(*			
	RAFALOS
	Rafał Osajda		19.09.2025		TC 4024.66
	Komponent bazowy dla elementów prostych
*)
FUNCTION_BLOCK FB_BaseComponent EXTENDS FB_BaseLoggerElement IMPLEMENTS ITF_BaseComponent, ITF_BaseComponent_HMI_Connector
VAR
	cmdReset						: FB_BaseCommand;
	cmdParametersCreate				: FB_BaseCommand;
	cmdParametersRestoreToDefault	: FB_BaseCommand;
	
	
END_VAR
VAR PERSISTENT
	stParameters					: ST_Parameters;
END_VAR

(*			
	RafalOS
	Rafał Osajda		27.03.2025		TC 4024.66
	Obsluga bledow sprawdzanie czy jakis blad sie nei pojawil i ustawienie stanu lub wylaczenie
*)
METHOD PUBLIC ExecuteEveryCycle_Error
VAR_INPUT
END_VAR
END_METHOD

(*			
	RafalOS
	Rafał Osajda		27.03.2025		TC 4024.66
	Wywolanie co cykl operacji 
*)
METHOD PUBLIC ExecuteEveryCycle_Operation
VAR_INPUT
END_VAR
IF (THIS^.cmdReset.OperationExecute ()) THEN
	THIS^.cmdReset.Operation (bIN		:= THIS^.ResetOperation ());
END_IF

IF (THIS^.cmdParametersCreate.OperationExecute ()) THEN
	THIS^.cmdParametersCreate.Operation (bIN := THIS^.ParameterCreateTable ());
END_IF

IF (THIS^.cmdParametersRestoreToDefault.OperationExecute ()) THEN
	THIS^.cmdParametersRestoreToDefault.Operation (bIN	:= THIS^.ParameterRestoreDefaultValueAll ());
END_IF
END_METHOD

(*			
	RafalOS
	Rafał Osajda		27.03.2025		TC 4024.66
	Aktualizacja flag 
*)
METHOD PUBLIC ExecuteEveryCycle_Status
VAR_INST
END_VAR
END_METHOD

(*			
	RafalOS
	Rafał Osajda		27.03.2025		TC 4024.66
	Testowanie czy nei pojawil sie jakis rozkaz i uruchomienie odpowiednich operacji
*)
METHOD PUBLIC ExecuteEveryCycle_Test
VAR_INPUT
END_VAR
THIS^.cmdReset.Test ();
THIS^.cmdParametersCreate.Test ();
THIS^.cmdParametersRestoreToDefault.Test ();
END_METHOD

METHOD FB_init : BOOL
VAR_INPUT
	bInitRetains : BOOL; // if TRUE, the retain variables are initialized (warm start / cold start)
	bInCopyCode : BOOL;  // if TRUE, the instance afterwards gets moved into the copy code (online change)
END_VAR
THIS^.stIdentifier.eType			:= E_BaseElementType.eComponent;
END_METHOD

(*			
	RafalOS
	Rafał Osajda		03.10.2025		TC 4024.66
	
*)
METHOD PUBLIC FirstCycle : BOOL
VAR_INPUT
END_VAR
FirstCycle				:= SUPER^.FirstCycle ();
END_METHOD

METHOD GetITFComponent : ITF_BaseComponent
VAR_INPUT
END_VAR
GetITFComponent		:= THIS^;
END_METHOD

METHOD GetITFControlElement : ITF_BaseControlElement
VAR_INPUT
END_VAR
GetITFControlElement	:= null;
END_METHOD

METHOD GetITFGroupElement : ITF_BaseGroupElement
VAR_INPUT
END_VAR
GetITFGroupElement	:= null;
END_METHOD

METHOD GetITFTopElement : ITF_BaseTopElement
VAR_INPUT
END_VAR
GetITFTopElement		:= null;
END_METHOD

(*			
	RafalOS
	Rafał Osajda		07.10.2025		TC 4024.66
	Dodpisywanie się do listy logera
*)
METHOD PUBLIC JoinTheLogger : BOOL
VAR_INPUT
END_VAR
IF (THIS^.bIsValidCommonData) THEN
	IF (THIS^.refstCommonData.itfLogger.AddItem (itfItem := THIS^) > 0 ) THEN
		JoinTheLogger		:= TRUE;
	END_IF
END_IF
END_METHOD

(*			
	RafalOS
	Rafał Osajda		26.03.2025		TC 4024.66
	Dodawanie parametru do elementu wykonawczego - metode wywołać przy pierwszym uruchomieniu programu by wgrać parametry do pamięci
	później używać tylko edycji lub przywracania wartości domyślnych
*)
METHOD PUBLIC ParameterAdd : BOOL
VAR_INPUT
	stParameter			: ST_BaseDescriptor;
END_VAR
IF (THIS^.stParameters.uiNumber + 1 <= TO_UINT (GVL_BaseConstans.MAX_NUMBER_OF_PARAMETERS)) THEN
	THIS^.stParameters.uiNumber 		:= THIS^.stParameters.uiNumber + 1;
	THIS^.stParameters.arrRow [THIS^.stParameters.uiNumber] 	:= stParameter;
	ParameterAdd				:= TRUE;
ELSE
	ParameterAdd				:= FALSE;
END_IF
END_METHOD

(*			
	RafalOS
	Rafał Osajda		26.03.2025		TC 4024.66
	Modyfikuje wartość domyślną w istniejącym parametrze - true jak się zmiana udała
*)
METHOD PUBLIC ParameterCorrectDefaultValue : BOOL
VAR_INPUT
	uiNumber			: UINT;
	rValue				: REAL;
END_VAR
IF (uiNumber > 0 AND uiNumber <= THIS^.stParameters.uiNumber) THEN
	IF (rValue >= THIS^.GetMinFrom (stIN := THIS^.stParameters.arrRow [uiNumber]) AND
		rValue <= THIS^.GetMaxFrom (stIN := THIS^.stParameters.arrRow [uiNumber])) THEN
		THIS^.SetDefaultValueIn (stIN := THIS^.stParameters.arrRow [uiNumber], rDefaultValue	:= rValue);
		ParameterCorrectDefaultValue		:= TRUE;
	ELSE
		ParameterCorrectDefaultValue		:= FALSE;
	END_IF
ELSE
	ParameterCorrectDefaultValue		:= FALSE;
END_IF
END_METHOD

METHOD PUBLIC ParameterCorrectName : BOOL
VAR_INPUT
	eLocation					: E_BaseLocation;
	uiNumberOfParameter			: UINT;
	wsDescription				: WSTRING;
END_VAR
THIS^.SetTextIn (
	stIN 			:= THIS^.stParameters.arrRow [uiNumberOfParameter],
	eLocation		:= eLocation,
	wsDescription	:= wsDescription
);
END_METHOD

(*			
	RafalOS
	Rafał Osajda		26.03.2025		TC 4024.66
	Modyfikuje wartość w istniejącym parametrze - true jak się zmiana udała
*)
METHOD PUBLIC ParameterCorrectValue : BOOL
VAR_INPUT
	uiNumber			: UINT;
	rValue				: REAL;
END_VAR
IF (uiNumber > 0 AND uiNumber <= THIS^.stParameters.uiNumber) THEN
	IF (rValue <= THIS^.GetMaxFrom (stIN := THIS^.stParameters.arrRow [uiNumber]) AND
		rValue >= THIS^.GetMinFrom (stIN := THIS^.stParameters.arrRow [uiNumber]) ) THEN
		THIS^.SetValueIn (
			stIN		:= THIS^.stParameters.arrRow [uiNumber],
			rValue		:= rValue
		);
		ParameterCorrectValue		:= TRUE;
	ELSE
		ParameterCorrectValue		:= FALSE;
	END_IF
ELSE
	ParameterCorrectValue		:= FALSE;
END_IF
END_METHOD

(*			
	RafalOS
	Rafał Osajda		31.03.2025		TC 4024.66
	Metoda wymazująca dotychczasowe dane z tablicy parametrów i przypisująca je od nowa
*)
METHOD PROTECTED ParameterCreateTable : BOOL
VAR_INPUT
END_VAR
MEMSET (
	destAddr			:= ADR (THIS^.stParameters.arrRow),
	fillByte			:= 0,
	n					:= SIZEOF (THIS^.stParameters.arrRow)
);
THIS^.stParameters.uiNumber	:= 0;

ParameterCreateTable := TRUE;
END_METHOD

METHOD PUBLIC ParameterGet : ST_BaseDescriptor
VAR_INPUT
	uiNumer				: UINT;
END_VAR
ParameterGet			:= THIS^.stParameters.arrRow [uiNumer];
END_METHOD

(*			
	RafalOS
	Rafał Osajda		26.03.2025		TC 4024.66
	Zwraca wartosc domyslna
*)
METHOD PUBLIC ParameterGetDefaultValue : REAL
VAR_INPUT
	uiNumber				: UINT;
END_VAR
IF (uiNumber > 0 AND uiNumber <= THIS^.stParameters.uiNumber) THEN
	ParameterGetDefaultValue			:= THIS^.GetDefaultValueFrom (stIN :=  THIS^.stParameters.arrRow [uiNumber]);
ELSE
	ParameterGetDefaultValue			:= 0;
END_IF
END_METHOD

(*			
	RafalOS
	Rafał Osajda		26.03.2025		TC 4024.66
	Zwraca wartość MAX
*)
METHOD PUBLIC ParameterGetMax : REAL
VAR_INPUT
	uiNumber				: UINT;
END_VAR
IF (uiNumber > 0 AND uiNumber <= THIS^.stParameters.uiNumber) THEN
	ParameterGetMax			:= THIS^.GetMaxFrom (stIN :=  THIS^.stParameters.arrRow [uiNumber]);
ELSE
	ParameterGetMax			:= 0;
END_IF
END_METHOD

(*			
	RafalOS
	Rafał Osajda		26.03.2025		TC 4024.66
	Zwraca wartość MIN
*)
METHOD PUBLIC ParameterGetMin : REAL
VAR_INPUT
	uiNumber				: UINT;
END_VAR
IF (uiNumber >= 0 AND uiNumber <= THIS^.stParameters.uiNumber) THEN
	ParameterGetMin			:= THIS^.GetMinFrom (stIN := THIS^.stParameters.arrRow [uiNumber]);
ELSE
	ParameterGetMin			:= 0;
END_IF
END_METHOD

METHOD PUBLIC ParameterGetNumberOfAdded : UINT
VAR_INPUT
END_VAR
ParameterGetNumberOfAdded			:= THIS^.stParameters.uiNumber;
END_METHOD

(*			
	RafalOS
	Rafał Osajda		26.03.2025		TC 4024.66
	Zwraca jednostke
*)
METHOD PUBLIC ParameterGetUnit : STRING(6)
VAR_INPUT
	uiNumber				: uINT;
END_VAR
IF (uiNumber > 0 AND uiNumber <= THIS^.stParameters.uiNumber) THEN
	ParameterGetUnit			:= THIS^.GetUnitFrom (stIN :=  THIS^.stParameters.arrRow [uiNumber]);
ELSE
	ParameterGetUnit			:= '';
END_IF
END_METHOD

(*			
	RafalOS
	Rafał Osajda		26.03.2025		TC 4024.66
	Zwraca wartość
*)
METHOD PUBLIC ParameterGetValue : REAL
VAR_INPUT
	uiNumber				: UINT;
END_VAR
IF (uiNumber > 0 AND uiNumber <= THIS^.stParameters.uiNumber) THEN
	ParameterGetValue			:= THIS^.GetValueFrom (stIN := THIS^.stParameters.arrRow [uiNumber]);
ELSE
	ParameterGetValue			:= 0;
END_IF
END_METHOD

(*			
	RafalOS
	Rafał Osajda		26.03.2025		TC 4024.66
	Modyfikacja istniejącego parametra jako przypisanie nowego deskryptora
*)
METHOD PUBLIC ParameterModify : BOOL
VAR_INPUT
	uiNumber			: UINT;
	stParameter			: ST_BaseDescriptor;
END_VAR
IF (uiNumber > 0 AND uiNumber <= THIS^.stParameters.uiNumber) THEN
	THIS^.stParameters.arrRow [uiNumber]	:= 	stParameter;
	ParameterModify		:= TRUE;
ELSE
	ParameterModify		:= FALSE;
END_IF
END_METHOD

METHOD PUBLIC ParameterRestoreDefaultValue : BOOL
VAR_INPUT
	uiNumber		: UINT;
END_VAR
IF (uiNumber > 0 AND uiNumber <= THIS^.stParameters.uiNumber) THEN
	THIS^.SetValueIn (stIN := THIS^.stParameters.arrRow [uiNumber], rValue := THIS^.GetDefaultValueFrom (stIN := THIS^.stParameters.arrRow [uiNumber]));
	ParameterRestoreDefaultValue	:= TRUE;
ELSE
	ParameterRestoreDefaultValue	:= FALSE;
END_IF
END_METHOD

METHOD PROTECTED ParameterRestoreDefaultValueAll : BOOL
VAR_INPUT
END_VAR

VAR
	iI					: INT;
	bResult				: bool;
END_VAR
bResult					:= TRUE;
FOR iI := 1 TO TO_INT (THIS^.stParameters.uiNumber) DO 
	bResult				:= bResult AND THIS^.ParameterRestoreDefaultValue (uiNumber := TO_UINT (iI));
END_FOR
END_METHOD

(*			
	RafalOS
	Rafał Osajda		04.05.2025		TC 4024.66
	Skasowanie i utworzenie tablicy parametrów od nowa 
*)
METHOD PUBLIC ParametersCreate : BOOL
THIS^.cmdParametersCreate.Execute ();
END_METHOD

(*			
	RafalOS
	Rafał Osajda		04.05.2025		TC 4024.66
	Przywrocenie parametrow - in na false to tylko ten element true razem z podelementami
*)
METHOD PUBLIC ParameterSetToDefault : BOOL
THIS^.cmdParametersRestoreToDefault.Execute ();
END_METHOD

METHOD PUBLIC Reset : BOOL
VAR_INPUT
END_VAR
THIS^.cmdReset.Execute ();
END_METHOD

METHOD PUBLIC ResetGetBusy : BOOL
VAR_INPUT
END_VAR
ResetGetBusy		:= THIS^.cmdReset.IsBusy ();
END_METHOD

METHOD PUBLIC ResetGetStatus : BOOL
VAR_INPUT
END_VAR
ResetGetStatus			:= THIS^.cmdReset.IsStatus ();
END_METHOD

METHOD PROTECTED ResetOperation : BOOL
VAR_INPUT
END_VAR


ResetOperation			:= FALSE;
END_METHOD

END_FUNCTION_BLOCK

(* stored: Version 1.1.0.1
   POU FB_BaseComponent: Id {87e0f050-2d49-0545-1d2d-1d8cc43d61c2}, SpecialFunc None
   Folder ITF_BaseComponent: Id {b16f93e1-934e-0805-383f-d97d810c646e}
   Folder ITF_DecoratedElement: Id {41521ef6-d598-047e-2c22-8e73616ee08c}
   Folder Parameter: Id {51f1d98c-bdeb-0f9b-3843-7bd8ef234ec3}
   Method ExecuteEveryCycle_Error: Id {d0f95f17-dd99-064c-15eb-b6a90cafd74d}
   Method ExecuteEveryCycle_Operation: Id {513159e8-2790-0493-315a-cd955c8d31c5}
   Method ExecuteEveryCycle_Status: Id {4211d7fe-e3a3-005a-3d2b-874c421b8ff4}
   Method ExecuteEveryCycle_Test: Id {4131c775-8fd3-0b9a-02c8-9e9a0a682b52}
   Method FB_init: Id {f6b4fcc3-c3c0-0af2-28d1-79ccbb610da2}
   Method FirstCycle: Id {59d66408-2df1-04a5-240d-93e8399a3b7e}
   Method GetITFComponent: Id {33e10c5b-120b-0f78-06cf-170e49fa6c9a}
   Method GetITFControlElement: Id {9af90360-abec-083a-18a8-2f7d8868516c}
   Method GetITFGroupElement: Id {aa64e9b4-f847-0695-3ed1-9b7a5b38ab92}
   Method GetITFTopElement: Id {20a46a89-89ab-043b-0602-3d56a5db1953}
   Method JoinTheLogger: Id {c36b1ddd-e3f3-0707-2e1b-24a85c94c962}
   Method ParameterAdd: Id {0bbb0fac-f279-0b70-341a-ed0caf27ff48}
   Method ParameterCorrectDefaultValue: Id {ea5554ac-46a4-0090-2247-7c38cc711c17}
   Method ParameterCorrectName: Id {cc4d8743-c51f-0c67-0f5d-3ed9379dd6b6}
   Method ParameterCorrectValue: Id {7c6db1a2-5e76-0e89-3719-a5d4c4278993}
   Method ParameterCreateTable: Id {5c2e0dd4-2d80-0a33-06c5-97040748aaef}
   Method ParameterGet: Id {d8c0108f-8a5a-0b99-2668-1679555db078}
   Method ParameterGetDefaultValue: Id {988eb6f3-0732-0567-16cf-3de68eec0a9a}
   Method ParameterGetMax: Id {5c28c07f-b14c-0760-37a9-6dacdce80dc2}
   Method ParameterGetMin: Id {89312f05-57f5-0184-360c-08b141ef26e1}
   Method ParameterGetNumberOfAdded: Id {74c11ec2-a556-0bd7-3162-91c4a03b75e5}
   Method ParameterGetUnit: Id {bb9b2833-f611-0468-2fc2-8a7dc470b3d3}
   Method ParameterGetValue: Id {bc97081f-e202-05b7-3cad-6b67ebf2409d}
   Method ParameterModify: Id {e578fbe4-e52c-0213-244a-972cbc85a1ef}
   Method ParameterRestoreDefaultValue: Id {139a3102-43d8-0081-0eb2-892be4ec2d31}
   Method ParameterRestoreDefaultValueAll: Id {0026bcd4-2ada-0a85-0709-2aa759eab8a8}
   Method ParametersCreate: Id {c946a0bf-5c4e-0c5c-0419-301bd87e62bd}
   Method ParameterSetToDefault: Id {3020fada-bbb7-04bb-27d1-a0f7481f168e}
   Method Reset: Id {c0bf4177-e97f-089b-34b4-b48fadeb74cc}
   Method ResetGetBusy: Id {3b84d943-6444-09e4-127e-9583cbeebff0}
   Method ResetGetStatus: Id {d861273e-29d7-0151-12ed-78079fcd5e28}
   Method ResetOperation: Id {2d760c90-c43b-0af4-3d18-a1d7b05cea9c} *)
